FUNCTION F_HMI_HEALTH_TO_COLOR : T_HMI_COLORS
VAR_IN_OUT
    fbHealthStatus : FB_HMI_HEALTH_STATUS;
END_VAR
VAR_OUTPUT
END_VAR
VAR
END_VAR

IF fbHealthStatus.bGood THEN
    F_HMI_HEALTH_TO_COLOR.fg := E_HMI_COLORS.BLACK;
    F_HMI_HEALTH_TO_COLOR.bg := E_HMI_COLORS.GREEN;
ELSIF fbHealthStatus.bBad THEN
	F_HMI_HEALTH_TO_COLOR.fg := E_HMI_COLORS.WHITE;
	F_HMI_HEALTH_TO_COLOR.bg := E_HMI_COLORS.RED;
ELSIF fbHealthStatus.bWarning THEN
	F_HMI_HEALTH_TO_COLOR.fg := E_HMI_COLORS.WHITE;
	F_HMI_HEALTH_TO_COLOR.bg := E_HMI_COLORS.ORANGE;
ELSE
	F_HMI_HEALTH_TO_COLOR.fg := E_HMI_COLORS.BLACK;
	F_HMI_HEALTH_TO_COLOR.bg := E_HMI_COLORS.GRAY;
END_IF

END_FUNCTION

(* stored: Version 1.1.0.1, ProductVersion 3.1.4024.14
   POU F_HMI_HEALTH_TO_COLOR: Id {299e323c-264e-4374-b012-e299b5a3bc8a}, SpecialFunc None *)
